// TIA Portal V19 export
DATA_BLOCK "ALARMS_DB"   // DB116
{ S7_Optimized_Access := 'FALSE' }
   VAR
      "EMERGENCY STOP" : Bool;
      "PHASE FAIL" : Bool;
      "AIR PRESSURE FAIL" : Bool;
      "REGENRATION OVER" : Bool;
      "LT-1 LOW LOW" : Bool;
      "LT-1 HIGH HIGH" : Bool;
      "LS-5 LOW" : Bool;
      "PS-1 LOW" : Bool;
      "PS-2 LOW" : Bool;
      "LT-2 HIGH HIGH" : Bool;
   END_VAR
BEGIN
END_DATA_BLOCK
